// TIA Portal V19 export
TYPE "LEXCHANGETRAY_typeSr1000ProfinetTelegram_latchandErrorClearControlBits"
// stored: Access Published
   STRUCT
      controlByte : Byte;
      resultDataLatch : Bool;
      errorClear : Bool;
   END_STRUCT;
END_TYPE
